Yaskawa INFORM job: TWIN_5340_0ST_RAMA_PRZ_OBR1_POM.JBI

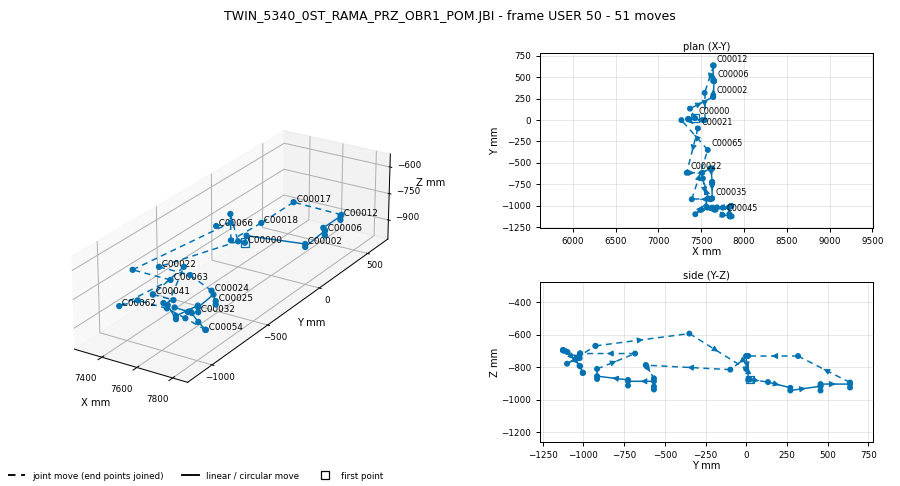
[picture p0: tool path of TWIN_5340_0ST_RAMA_PRZ_OBR1_POM.JBI in frame USER 50, 51 of 51 moves have a stored position in this frame; points joined in program order, loops and branches not executed]
/JOB
//NAME TWIN_5340_0ST_RAMA_PRZ_OBR1_POM
///FOLDERNAME 02-SKRZYNIE_JOBS
//POS
///NPOS 67,67,0,9,0,0
///USER 50
///TOOL 0
///POSTYPE USER
///RECTAN
///RCONF 1,0,0,0,0,0,0,0,0,0,0,0,0,0,0,0,0,0,0,0,0,0,0,0
C00000=7427.866,22.110,-875.338,0.7797,5.2883,0.7525
C00001=7368.857,133.592,-891.357,4.8365,6.9903,8.6973
///RCONF 0,0,0,0,0,0,0,0,0,0,0,0,0,0,0,0,0,0,0,0,0,0,0,0
C00002=7639.863,270.867,-926.395,13.5839,-33.1983,13.1947
C00003=7639.853,270.876,-946.071,13.5848,-33.1976,13.1942
C00004=7639.846,270.881,-942.884,13.5863,-33.1973,13.1931
C00005=7671.364,270.875,-942.909,13.5851,-33.1954,13.1944
C00006=7650.482,456.002,-916.839,13.5844,-33.1961,13.1959
C00007=7650.482,456.002,-916.839,13.5844,-33.1961,13.1959
C00008=7650.451,455.996,-947.503,13.5859,-33.1931,13.1943
C00009=7650.478,455.991,-943.413,13.5875,-33.1948,13.1918
C00010=7675.927,455.999,-943.433,13.5864,-33.1946,13.1935
C00011=7640.276,455.996,-903.574,13.5846,-33.1967,13.1949
C00012=7640.287,637.284,-903.553,13.5865,-33.1975,13.1927
C00013=7640.279,637.279,-928.515,13.5923,-33.1955,13.1860
C00014=7640.284,637.264,-924.743,13.5865,-33.1971,13.1919
C00015=7681.222,637.270,-924.755,13.5900,-33.1951,13.1887
C00016=7645.873,637.254,-894.160,13.5893,-33.1969,13.1883
C00017=7539.942,318.049,-731.449,13.5900,-33.1963,13.1869
C00018=7539.941,-1.151,-731.443,13.5934,-33.1961,13.1829
///RCONF 1,0,0,0,0,0,0,0,0,0,0,0,0,0,0,0,0,0,0,0,0,0,0,0
C00019=7350.000,12.009,-876.948,0.1408,4.3424,0.4590
C00020=7346.874,12.003,-730.531,0.1396,4.3422,0.4627
C00021=7461.700,-97.675,-814.930,5.9111,-6.8047,-23.4203
///RCONF 0,0,0,0,0,0,0,0,0,0,0,0,0,0,0,0,0,0,0,0,0,0,0,0
C00022=7330.504,-616.291,-787.560,-6.3273,-30.3234,-48.5706
C00023=7511.957,-616.291,-787.560,-6.3273,-30.3234,-48.5706
C00024=7603.003,-566.694,-868.189,-6.3274,-30.3238,-48.5709
C00025=7626.994,-566.690,-918.795,-6.3245,-30.3240,-48.5747
C00026=7626.962,-566.683,-941.026,-6.3207,-30.3222,-48.5804
C00027=7626.957,-566.651,-937.111,-6.3208,-30.3198,-48.5793
C00028=7673.428,-566.638,-937.170,-6.3198,-30.3163,-48.5812
C00029=7614.240,-566.649,-886.476,-6.3223,-30.3151,-48.5800
C00030=7628.645,-725.860,-886.466,-6.3211,-30.3161,-48.5819
C00031=7628.666,-725.848,-917.814,-6.3177,-30.3167,-48.5849
C00032=7628.647,-725.839,-912.981,-6.3161,-30.3156,-48.5874
C00033=7674.239,-725.840,-912.992,-6.3179,-30.3146,-48.5858
C00034=7627.183,-725.833,-877.944,-6.3161,-30.3152,-48.5868
C00035=7627.215,-915.908,-855.038,-6.3161,-30.3163,-48.5849
C00036=7627.213,-915.915,-877.878,-6.3162,-30.3169,-48.5852
C00037=7627.220,-915.900,-872.306,-6.3179,-30.3161,-48.5831
C00038=7675.637,-915.917,-872.316,-6.3187,-30.3156,-48.5842
C00039=7581.078,-915.910,-810.557,-6.3191,-30.3155,-48.5830
///RCONF 1,0,0,0,1,0,0,0,0,0,0,0,0,0,0,0,0,0,0,0,0,0,0,0
C00040=7519.943,-682.446,-716.060,47.7750,-2.1777,-137.5865
///RCONF 1,0,0,0,0,0,0,0,0,0,0,0,0,0,0,0,0,0,0,0,0,0,0,0
C00041=7568.741,-1020.042,-716.037,47.7758,-2.1774,-137.5877
///RCONF 0,0,0,0,0,0,0,0,0,0,0,0,0,0,0,0,0,0,0,0,0,0,0,0
C00042=7568.723,-1020.050,-716.048,63.5786,15.1002,-135.5502
C00043=7684.087,-1020.087,-716.287,63.5596,15.0824,-135.5554
C00044=7629.012,-1022.497,-744.338,76.9005,26.8308,-122.4425
C00045=7748.994,-1108.058,-702.116,77.1581,27.0674,-135.7350
C00046=7835.563,-1121.962,-696.031,82.0270,31.2593,-137.0869
C00047=7835.573,-1140.704,-696.017,82.0277,31.2621,-137.0871
C00048=7835.564,-1125.279,-696.024,82.0278,31.2616,-137.0870
C00049=7835.542,-1125.282,-696.043,82.3175,31.7788,-128.8636
C00050=7855.098,-1125.253,-696.030,82.3176,31.7796,-128.8622
C00051=7867.092,-1125.250,-696.152,82.3067,31.7743,-128.8681
C00052=7828.640,-1097.437,-706.872,82.3062,31.7737,-128.8691
///RCONF 0,0,0,0,1,0,0,0,0,0,0,0,0,0,0,0,0,0,0,0,0,0,0,0
C00053=7821.545,-1020.324,-793.634,46.2888,11.3440,-105.7987
C00054=7850.544,-1003.323,-834.254,46.2910,11.3478,-105.7983
C00055=7850.593,-1003.284,-855.210,46.2918,11.3479,-105.7928
C00056=7850.544,-1003.323,-834.254,46.2910,11.3478,-105.7983
C00057=7866.302,-1003.315,-834.268,46.2895,11.3486,-105.7987
C00058=7850.544,-1003.323,-834.254,46.2910,11.3478,-105.7983
///RCONF 0,0,0,0,0,0,0,0,0,0,0,0,0,0,0,0,0,0,0,0,0,0,0,0
C00059=7751.828,-1023.584,-791.330,53.9458,8.0938,-106.3571
C00060=7665.622,-1048.224,-752.179,61.6283,6.0169,-112.0769
C00061=7501.147,-1048.224,-752.179,61.6283,6.0169,-112.0769
C00062=7431.124,-1100.346,-778.577,-43.9463,-22.1147,3.1992
C00063=7605.796,-925.674,-669.082,-44.6202,-26.9485,11.2628
C00064=7389.781,-925.674,-669.082,-44.6202,-26.9485,11.2628
C00065=7576.917,-349.464,-593.545,-31.3975,-43.7406,20.7512
///RCONF 1,0,0,0,0,0,0,0,0,0,0,0,0,0,0,0,0,0,0,0,0,0,0,0
C00066=7268.753,-0.585,-810.777,7.4227,29.9022,-148.3766
///RCONF 0,0,0,0,0,0,0,0,0,0,0,0,0,0,0,0,0,0,0,0,0,0,0,0
BC00000=6131.609
BC00001=6231.609
BC00002=6231.609
BC00003=6231.609
BC00004=6231.609
BC00005=6231.609
BC00006=6231.609
BC00007=6231.609
BC00008=6231.609
BC00009=6231.609
BC00010=6231.609
BC00011=6231.609
BC00012=6231.609
BC00013=6231.609
BC00014=6231.609
BC00015=6231.609
BC00016=6231.609
BC00017=6231.609
BC00018=6231.609
BC00019=6132.996
BC00020=5940.084
BC00021=6107.541
BC00022=6231.609
BC00023=6413.063
BC00024=6413.063
BC00025=6413.063
BC00026=6413.063
BC00027=6413.063
BC00028=6413.063
BC00029=6413.063
BC00030=6413.063
BC00031=6413.063
BC00032=6413.063
BC00033=6413.063
BC00034=6413.063
BC00035=6413.063
BC00036=6413.063
BC00037=6413.063
BC00038=6413.063
BC00039=6413.063
BC00040=6260.553
BC00041=6260.553
BC00042=6260.553
BC00043=6376.118
BC00044=6448.288
BC00045=6557.032
BC00046=6557.032
BC00047=6557.032
BC00048=6557.032
BC00049=6557.032
BC00050=6557.032
BC00051=6557.038
BC00052=6557.038
BC00053=6557.038
BC00054=6557.038
BC00055=6557.038
BC00056=6557.038
BC00057=6557.038
BC00058=6557.038
BC00059=6494.392
BC00060=6399.125
BC00061=6234.649
BC00062=6234.649
BC00063=6234.649
BC00064=6018.634
BC00065=5794.475
BC00066=5960.552
///POSTYPE BASE
P00006=-2.449,0.031,8.825,0.0000,0.0000,0.0000
P00021=6.550,-0.003,-5.735,0.0000,0.0000,0.0000
P00022=5.943,-0.018,-6.388,0.0000,0.0000,0.0000
P00023=7.025,-0.019,-7.168,0.0000,0.0000,0.0000
P00024=5.926,-0.047,-4.777,0.0000,0.0000,0.0000
P00025=1.385,-0.036,8.652,0.0000,0.0000,0.0000
P00026=0.001,0.024,7.658,0.0000,0.0000,0.0000
P00280=-0.761,-1.221,0.004,0.0000,0.0000,0.0000
///RCONF 0,0,0,0,1,0,0,0,0,0,0,0,0,0,0,0,0,0,0,0,0,0,0,0
P00290=-0.023,-0.050,5.560,0.0000,0.0000,0.0000
//INST
///DATE 2024/10/25 11:04
///ATTR SC,RW,RJ
////FRAME USER 50
///GROUP1 RB1,BS1
NOP
'.................
'.................
'.................
'DODAC PROG POMIARY RAMA PRZED
'.................
'.................
'.................
SFTOF
MOVJ C00000 BC00000 VJ=50.00
'W5L
MOVJ C00001 BC00001 VJ=30.00 PL=0
MOVL C00002 BC00002 V=166.7
REFP 3 C00003 BC00003
CALL JOB:SEARCH-R1
SET P0021 P0006
SFTON P0021
MOVL C00004 BC00004 V=166.7
REFP 3 C00005 BC00005
CALL JOB:SEARCH-R1
SET P0021 P0006
SFTON P0021
SFTOF
MOVL C00006 BC00006 V=166.7
'W6L
MOVL C00007 BC00007 V=166.7
REFP 3 C00008 BC00008
CALL JOB:SEARCH-R1
SET P0022 P0006
SFTON P0022
MOVL C00009 BC00009 V=166.7
REFP 3 C00010 BC00010
CALL JOB:SEARCH-R1
SET P0022 P0006
SFTON P0022
SFTOF
MOVL C00011 BC00011 V=166.7
'W6P
MOVL C00012 BC00012 V=333.3 PL=0
REFP 3 C00013 BC00013
CALL JOB:SEARCH-R1
SET P0023 P0006
SFTON P0023
MOVL C00014 BC00014 V=166.7
REFP 3 C00015 BC00015
CALL JOB:SEARCH-R1
SET P0023 P0006
SFTON P0023
SFTOF
MOVL C00016 BC00016 V=166.7
MOVJ C00017 BC00017 VJ=20.00
MOVJ C00018 BC00018 VJ=20.00
MOVJ C00019 BC00019 VJ=20.00
MOVJ C00020 BC00020 VJ=20.00
MOVJ C00021 BC00021 VJ=20.00
MOVJ C00022 BC00022 VJ=20.00
MOVJ C00023 BC00023 VJ=20.00
MOVJ C00024 BC00024 VJ=40.00
MOVL C00025 BC00025 V=333.3 PL=0
REFP 3 C00026 BC00026
CALL JOB:SEARCH-R1
SET P0024 P0006
SFTON P0024
MOVL C00027 BC00027 V=166.7
REFP 3 C00028 BC00028
CALL JOB:SEARCH-R1
SET P0024 P0006
SFTON P0024
SFTOF
MOVL C00029 BC00029 V=166.7
MOVL C00030 BC00030 V=333.3 PL=0
REFP 3 C00031 BC00031
CALL JOB:SEARCH-R1
SET P0025 P0006
SFTON P0025
MOVL C00032 BC00032 V=166.7
REFP 3 C00033 BC00033
CALL JOB:SEARCH-R1
SET P0025 P0006
SFTON P0025
SFTOF
MOVL C00034 BC00034 V=166.7
MOVL C00035 BC00035 V=333.3 PL=0
REFP 3 C00036 BC00036
CALL JOB:SEARCH-R1
SET P0026 P0006
SFTON P0026
MOVL C00037 BC00037 V=166.7
REFP 3 C00038 BC00038
CALL JOB:SEARCH-R1
SET P0026 P0006
SFTON P0026
SFTOF
MOVL C00039 BC00039 V=166.7
MOVJ C00040 BC00040 VJ=40.00
MOVJ C00041 BC00041 VJ=40.00
MOVJ C00042 BC00042 VJ=40.00
MOVJ C00043 BC00043 VJ=40.00
MOVJ C00044 BC00044 VJ=40.00
MOVJ C00045 BC00045 VJ=40.00
MOVL C00046 BC00046 V=250.0
REFP 3 C00047 BC00047
CALL JOB:SEARCH-R1
SET P0280 P0006
SFTON P0280
MOVL C00048 BC00048 V=166.7
MOVL C00049 BC00049 V=250.0
MOVL C00050 BC00050 V=166.7
REFP 3 C00051 BC00051
CALL JOB:SEARCH-R1
SET P0280 P0006
MOVL C00052 BC00052 V=166.7
SFTOF
MOVL C00053 BC00053 V=333.3
MOVL C00054 BC00054 V=166.7
REFP 3 C00055 BC00055
CALL JOB:SEARCH-R1
SET P0290 P0006
SFTON P0290
MOVL C00056 BC00056 V=166.7
REFP 3 C00057 BC00057
CALL JOB:SEARCH-R1
SET P0290 P0006
MOVL C00058 BC00058 V=166.7
MOVJ C00059 BC00059 VJ=20.00
SFTOF
MOVJ C00060 BC00060 VJ=30.00
MOVJ C00061 BC00061 VJ=40.00
MOVJ C00062 BC00062 VJ=40.00
MOVJ C00063 BC00063 VJ=40.00
MOVJ C00064 BC00064 VJ=40.00
MOVJ C00065 BC00065 VJ=50.00
MOVJ C00066 BC00066 VJ=50.00
END
